{attribute 'qualified_only'}
{attribute 'strict'}
TYPE E_DomeState :
(
	closed  := 0,
	open	:= 1,
	slewing := 2,
	error	:= 3
);
END_TYPE

(* stored: Version 1.1.0.1, ProductVersion 3.1.4024.15
   DUT E_DomeState: Id {c96709e9-bed9-4f1c-b47d-382f9c9b4e8c} *)
